{attribute 'qualified_only'}
VAR_GLOBAL
	bDigital_Inputs AT %I* : ARRAY[1..8] OF BOOL;
	bDigital_Outputs AT %Q* : ARRAY[1..8] OF BOOL;
END_VAR

(* stored: Version 1.1.0.1, ProductVersion 3.1.4024.12
   GVL GVL: Id {d5fa82fe-a284-4b51-80a9-8ff9bfa33216} *)
